// TIA Portal V16 export
// export: Created 2021-08-10T09:05:00.3691749Z, ExportSetting WithDefaults, WithReadOnly, DisplayName Totally Integrated Automation Portal, DisplayVersion V16, DisplayName TIA Portal Version Control Interface, DisplayVersion V16, DisplayName TIA Portal Openness, DisplayVersion V16, DisplayName TIA Portal Teamcenter Gateway, DisplayVersion V16, DisplayName SINAMICS Startdrive Advanced, DisplayVersion V16, DisplayName SINAMICS Startdrive G130, G150, S120, S150, SINAMICS MV, S210, DisplayVersion V16, DisplayName SINAMICS Startdrive G110M, G120, G120C, G120D, G120P, DisplayVersion V16, DisplayName STEP 7 Professional, DisplayVersion V16, DisplayName STEP 7 Safety, DisplayVersion V16, DisplayName WinCC Unified SCADA Engineering System, DisplayVersion V16
FUNCTION_BLOCK "fbStepSequencer"   // FB185, SCL
TITLE = Step sequence controller
{ S7_Optimized_Access := 'TRUE' }
AUTHOR : Boris
VERSION : 4.0
// Modified by Ken Brey 2010-08-25 KLB.  Added Initialization inputs and logic.
// Modified by Ken Brey 2006-08-08 Removed initialization of inputs.  Initializing inputs doesn't do anything.  The input value if un-wired will be the last value
//                                   set for that input in a different call.  The initialized value in the declaration section does not set it back to default
//                                   if unwired.  Allways supply values for all inputs.
// Modified by Tim Jager 2005-12-13 no block Id in error message
// Modified by Boris: branched -> simplified version, no errors, no timeout; still have to use static memory for TON/CurStep (might be fixed later using in/out structure)
// Modified by Nick Shea:  2012-03-30 Re-instated step mode
// stored: AutoNumber false, CodeModifiedDate 2021-07-03T08:38:43.5995384Z, CompileDate 2021-07-03T08:38:43.5995384Z, CreationDate 2020-02-26T09:46:55.060709Z, DownloadWithoutReinit false, HandleErrorsWithinBlock false, InterfaceModifiedDate 2017-09-27T20:53:33.4400806Z, IsConsistent true, IsIECCheckEnabled false, IsKnowHowProtected false, ISMultiInstanceCapable true, IsRetainMemResEnabled false, IsWriteProtected false, LibraryConformanceStatus The object is library-conformant., LibraryType fbStepSequencer V 3.0.1, LibraryTypeVersionGuid beea64d7-3359-4773-b63d-f289c4512550, MemoryReserve 100, ModifiedDate 2021-07-03T08:38:43.5995384Z, ParameterModified 2016-08-14T20:38:38.9589289Z, PLCSimAdvancedSupport true, SetENOAutomatically true, StructureModified 2016-08-14T20:38:38.9704141Z, UDAEnableTagReadback false
   VAR_INPUT
      iInStep { ExternalAccessible := 'False'; ExternalVisible := 'False'; ExternalWritable := 'False'} : Int;   // Constant: current step required for the FB to run
      iInNextStep { ExternalAccessible := 'False'; ExternalVisible := 'False'; ExternalWritable := 'False'} : Int;   // Next step to go to if step is done
      bInStepDone { ExternalAccessible := 'False'; ExternalVisible := 'False'; ExternalWritable := 'False'} : Bool;   // if step done logic is true, then we move from IN_STEP to NEXT_STEP
      tInStepDelay { ExternalAccessible := 'False'; ExternalVisible := 'False'; ExternalWritable := 'False'} : Time;   // After the step done input is true, we wait for x seconds before moving to next
      bInStepMode { ExternalAccessible := 'False'; ExternalVisible := 'False'; ExternalWritable := 'False'} : Bool;   // Pause sequence at completion of current step
      bInStepAdvance { ExternalAccessible := 'False'; ExternalVisible := 'False'; ExternalWritable := 'False'} : Bool;   // If paused, trigger next step
      bInit { ExternalAccessible := 'False'; ExternalVisible := 'False'; ExternalWritable := 'False'} : Bool;
      iInitStep { ExternalAccessible := 'False'; ExternalVisible := 'False'; ExternalWritable := 'False'} : Int;
   END_VAR
   VAR_OUTPUT
      bOutEnterEvent { ExternalAccessible := 'False'; ExternalVisible := 'False'; ExternalWritable := 'False'} : Bool;
      bOutExitEvent { ExternalAccessible := 'False'; ExternalVisible := 'False'; ExternalWritable := 'False'} : Bool;
      bOutPaused { ExternalAccessible := 'False'; ExternalVisible := 'False'; ExternalWritable := 'False'} : Bool;   // Sequence is currently paused.
      iOutCurrentStep { ExternalAccessible := 'False'; ExternalVisible := 'False'; ExternalWritable := 'False'} : Int;   // output current step
   END_VAR
   VAR
      TON_StepDelay { ExternalAccessible := 'False'; ExternalVisible := 'False'; ExternalWritable := 'False'; S7_SetPoint := 'True'} : TON_TIME;   // used to delay moving to the next step.
      iCurrentStep { ExternalAccessible := 'False'; ExternalVisible := 'False'; ExternalWritable := 'False'} : Int;   // Current step of the sequencer
      bAlreadyInThisStep { ExternalAccessible := 'False'; ExternalVisible := 'False'; ExternalWritable := 'False'} : Bool;
   END_VAR
   VAR_TEMP
      bNoStepDelay : Bool;   // step delay disabled
   END_VAR
BEGIN


   //*****************************************************************************************
   // INSTRUCTION SECTION
   ENO:=false; //init variables
   #bOutExitEvent :=false;
   #bOutEnterEvent:=false;

   IF (#iInStep=#iCurrentStep) THEN
       IF NOT #bAlreadyInThisStep THEN
           #bOutEnterEvent:=true;
           #bAlreadyInThisStep:=true;
       END_IF;
       IF #bInStepDone THEN
           //Run Step done Timer
           #TON_StepDelay(IN:=(TRUE),PT:=#tInStepDelay);

           //check if we are using a step delay
           #bNoStepDelay:= (#tInStepDelay<=T#0MS);

           //We can move to the next step if (STEP_DONE and StepDelay timer complete) 
           //  AND
           //(we are in step mode and the step advance is true, or if we are not in step mode 
           //  AND
           //It is not the first scan of this step
           IF ((#TON_StepDelay.Q OR #bNoStepDelay) AND (NOT #bInStepMode OR (#bInStepMode AND #bInStepAdvance)) AND NOT #bOutEnterEvent) THEN 
               #iCurrentStep   := #iInNextStep;   //move to next step
               //Reset Step done Timer
               #TON_StepDelay(IN:=(false),PT:=#tInStepDelay); 
               #bOutExitEvent:=true;
               #bAlreadyInThisStep:=false;
           END_IF;
       END_IF;
       #bOutPaused := #bInStepDone AND (#TON_StepDelay.Q OR #bNoStepDelay) AND (#bInStepMode AND NOT #bInStepAdvance);
       //Only set this if we are ok and in the right step
       ENO:= true;
   END_IF;
   IF (#bInit) THEN
       #iCurrentStep := #iInitStep;
       #bInit:=false;  //Clear so that if it is unwired on the next call, it is not run.
       #bAlreadyInThisStep:=false;
   END_IF;

   //Set output variables
   #iOutCurrentStep := #iCurrentStep;
   #tInStepDelay := T#0MS;
END_FUNCTION_BLOCK
